Staubli VAL3: create.pgx

public program create(string x_sEntryBoxName, string x_sMenu, num x_nFocused, num& x_nError[])
  local num l_i
  local num l_nPosX
  local num l_nPosY
  local num l_nError
  local string l_sCustomString
  local string l_sSubString
begin
  // This program initializes all the required data to create an entryBox on the
  // userPage
  //
  // Input Param
  //  x_sEntryBoxName : Name of the page library to load
  //  x_sMenu         : Menu to display at the bottom of the page.
  //  If x_sMenu is empty, use default menu specified in library (variable sMenu)
  //  x_nFocused : Item to be focused when page is first displayed
  //
  // Output Param
  //  x_Error : Error code
  //
  //Created 21/12/05                              CCUR
  //--------------------------------------------------------------
  // Load page library
  l_nError=pw:libLoad(x_sEntryBoxName)
  if (l_nError==0) or (l_nError==11)
    if len(x_sMenu)!=0
      pw:sMenu=x_sMenu
    endIf
    nNumOfLabel=size(pw:sLabel)
    nNumOfTxtBox=size(pw:sTxtBoxCaption)
    call pw:init(l_nError)
    if l_nError<0
      // Any internal error of the definition library are reported with code -2
      // However, a clear text is read an forwarded as an error of this library
      x_nError=-2
      // Prepare clear text error message
      call pw:getErrorMessage(l_sCustomString)
      l_sSubString=pw:libPath()
      call ut:addStrToString(sErrMsgList[-x_nError],sErrorMessage,"",l_sSubString)
      sErrorMessage=sErrorMessage+l_sCustomString
    else
      call _resizeData(nNumOfTxtBox,nNumOfLabel)
      nFocused=x_nFocused
    endIf
  else
    x_nError=1
    // Prepare clear text error message
    call ut:addStrToString(sErrMsgList[x_nError],sErrorMessage,"",x_sEntryBoxName)
    call ut:addNumToString(sErrorMessage,sErrorMessage,"*",l_nError)
  endIf
end
